(* IEC 61131-3 sources: CODESYS-IO-Visualization/CODESYS-IO-Visualization.fbsproj/Pi.device.xml.v3^/Plc Logic.plclogic.xml.v3^/Application.application.xml.v3^/Programs/3_Equipment, 1 file *)

(* ---- Main_Equipment.prg.st ---- *)
PROGRAM Main_Equipment
VAR
END_VAR

// ********** Base Equipment Code **********

// Pump 1 Inlet Valve: Site.Plant.Pump1.InletValve
Equip(Data := Site.Plant.Pump1.InletValve);

// Pump 1 Outlet Valve: Site.Plant.Pump1.OutletValve
Equip(Data := Site.Plant.Pump1.OutletValve);

// Pump 1 VFD: Site.Plant.Pump1.VFD
Equip(Data := Site.Plant.Pump1.VFD);
